// TwinCAT 3 PLC project LF_System_PLC
// ProgramVersion: 3.1.4026.20
// CompilerDefines: VISU_USEPROPERTYINFO
// libraries:
//   Tc2_Standard, * (Beckhoff Automation GmbH)
//   Tc2_System, * (Beckhoff Automation GmbH)
//   VisuSymbols, 4.5.0.0 (System)
// project tree:
//   DUTs/ Betriebszustand.TcDUT (not stored)
//   / GlobalTextList.TcGTLO, PlcTask.TcTTO (not stored), Visualization Manager.TcVMO (not stored)
//   POUs/Extruder/ FB_System_FlaschenFullstand.TcPOU (not stored), FB_System_Fullstand.TcPOU (not stored)
//   POUs/Förderband/ FB_System_CNV.TcPOU
//   POUs/ MAIN.TcPOU
//   POUs/Manipulator/ FB_System_LinAxis.TcPOU (not stored)
//   POUs/Vereinzelung/ FB_SpeicherRohr.TcPOU (not stored), FB_System_Vereinzelung.TcPOU (not stored)
//   VISUs/ Visualization.TcVIS
// (motion and I/O tree: see PLC project tempmodel)
// real-time tasks:
//   TASK PlcTask: cycle T#10ms, priority 21, ADS port 350
//   TASK PlcTask1: cycle T#10ms, priority 22, ADS port 351
//   TASK PlcTask2: cycle T#10ms, priority 20, ADS port 352
// variable links:
//   LF_System_PLC/LF_System_PLC Instance <-> NC-Task 1 SAF/Axes/BandAchse
//     PlcTask Inputs/MAIN.fIN_CnvPos <-> Outputs/ToPlc/ActPos
//   LF_System_PLC/LF_System_PLC Instance <-> NC-Task 1 SAF/Axes/Extruder1
//     PlcTask Inputs/MAIN.fIN_ExtPos1 <-> Outputs/ToPlc/ActPos
//   LF_System_PLC/LF_System_PLC Instance <-> NC-Task 1 SAF/Axes/Extruder2
//     PlcTask Inputs/MAIN.fIN_ExtPos2 <-> Outputs/ToPlc/ActPos
//   LF_System_PLC/LF_System_PLC Instance <-> NC-Task 1 SAF/Axes/Extruder3
//     PlcTask Inputs/MAIN.fIN_ExtPos3 <-> Outputs/ToPlc/ActPos
//   LF_System_PLC/LF_System_PLC Instance <-> PLC/PLC Instance
//     PlcTask Inputs/MAIN.bIN_Gripper <-> PlcTask Outputs/IFC_HW.bGripperClosed
//     PlcTask Inputs/MAIN.bIN_Stopper1 <-> PlcTask Outputs/IFC_HW.bBandHub1
//     PlcTask Inputs/MAIN.bIN_Stopper2 <-> PlcTask Outputs/IFC_HW.bBandHub2
//     PlcTask Inputs/MAIN.bIN_Stopper3 <-> PlcTask Outputs/IFC_HW.bBandHub3
//     PlcTask Inputs/MAIN.bIn_LedGreen <-> PlcTask Outputs/IFC_HW.bAmpelGrun
//     PlcTask Inputs/MAIN.bIn_LedRot <-> PlcTask Outputs/IFC_HW.bAmpelRot
//     PlcTask Inputs/MAIN.bIn_LedYellow <-> PlcTask Outputs/IFC_HW.bAmpelGelb
//     PlcTask Inputs/MAIN.bIn_Schleuse1_L1 <-> PlcTask Outputs/IFC_HW.bR1AKT1
//     PlcTask Inputs/MAIN.bIn_Schleuse1_L2 <-> PlcTask Outputs/IFC_HW.bR2AKT1
//     PlcTask Inputs/MAIN.bIn_Schleuse2_L1 <-> PlcTask Outputs/IFC_HW.bR1AKT2
//     PlcTask Inputs/MAIN.bIn_Schleuse2_L2 <-> PlcTask Outputs/IFC_HW.bR2AKT2
//     PlcTask Outputs/MAIN.bEnable <-> PlcTask Inputs/IFC_HW.bEnable
//     PlcTask Outputs/MAIN.bExecute <-> PlcTask Inputs/IFC_HW.bExecute
//     PlcTask Outputs/MAIN.bOUT_CnvNS{1..4} <-> PlcTask Inputs/IFC_HW.bBandSens{1..4}  (4 links)
//     PlcTask Outputs/MAIN.bOut_VereinzelungNS1 <-> PlcTask Inputs/IFC_HW.bEinzelSens1
//     PlcTask Outputs/MAIN.bOut_VereinzelungNS2 <-> PlcTask Inputs/IFC_HW.bEinzelSens2
//     PlcTask Outputs/MAIN.bOut_VereinzelungNS3 <-> PlcTask Inputs/IFC_HW.bEinzelSens3

// ---- POUs/Förderband/FB_System_CNV.TcPOU
FUNCTION_BLOCK FB_System_CNV
VAR_INPUT
	fPos : LREAL;
	bStopper1 : BOOL;
	bStopper2 : BOOL;
	bStopper3 : BOOL;
	bBottleDropped : BOOL; 
END_VAR
VAR_OUTPUT
	bNS1 : BOOL;
	bNS2 : BOOL;
	bNS3 : BOOL;
	bNS4 : BOOL;
	bBottleLeft : BOOL;
END_VAR
VAR
	fBottlePos : LREAL; // Reale Position der Flasche
	iBottlePos : LREAL; // Visualisierungs Position der Flaschen
	bBottleMoving : BOOL; // Flasche kann sich Bewegen, kein Stopper geschlossen und Stopper Pos erreicht
	fOffPos : LREAL; // OffsetPos nach Bewegungsfreigabe durch Stopper rückzug...
	rTrigBottleMoving : R_Trig;
	rTrigBottleDropped : R_Trig;
	fStopperPos1 : LREAL := 125.0;
	fStopperPos2 : LREAL := 250.0;
	fStopperPos3 : LREAL := 375.0;
	fStopperPos4 : LREAL := 630.0;; // Ende des Förderbandes
	onTimerCNVClear : TON;
	bBottleOnCNV : BOOL;
	bCNVisMoving : BOOL;
	fPosAlt : LReal;
END_VAR

onTimerCNVClear(PT := T#1S);
rTrigBottleMoving(CLK := bBottleMoving);
rTrigBottleDropped(CLK := bBottleDropped);
IF rTrigBottleDropped.Q THEN
	bBottleOnCNV := TRUE;
END_IF
// Flaschen Position bestimmen
IF rTrigBottleMoving.Q OR rTrigBottleDropped.Q THEN
	fOffPos := fPos-fBottlePos;
END_IF
IF bBottleMoving AND bBottleOnCNV THEN
	fBottlePos := fPos-fOffPos;
END_IF
// Skalierungsfunktion für fBottlePos zu iBottlePos (Real zu Visualisierung)

iBottlePos := TO_INT(fBottlePos * 0.7);

// Bewegungsfreigabe
IF NOT bStopper1 AND fBottlePos > fStopperPos1 - 2.0 AND fBottlePos < fStopperPos1 + 2.0 THEN
	bBottleMoving := FALSE;
ELSIF NOT bStopper2 AND fBottlePos > fStopperPos2 - 2.0 AND fbottlePos < fStopperPos2 + 2.0 THEN
	bBottleMoving := FALSE;
ELSIF NOT bStopper3 AND fBottlePos > fStopperPos3 - 2.0 AND fBottlePos < fStopperPos3 + 2.0 THEN
	bBottleMoving := FALSE;
ELSIF fBottlePos > fStopperPos4 - 1.0 THEN
	bBottleMoving := FALSE;
ELSE
	bBottleMoving := TRUE;
END_IF
// Sensor aktivierung
// bNS1
IF fBottlePos > fStopperPos1 - 15.0 AND fBottlePos < fStopperPos1 + 5.0 THEN
	bNS1 := TRUE;
ELSE
	bNS1 := FALSE;
END_IF
//bNS2
IF fBottlePos > fStopperPos2 - 15.0 AND fBottlePos < fStopperPos2 + 5.0 THEN
	bNS2 := TRUE;
ELSE
	bNS2 := FALSE;
END_IF
//bNS3
IF fBottlePos > fStopperPos3 - 15.0 AND fBottlePos < fStopperPos3 + 5.0 THEN
	bNS3 := TRUE;
ELSE
	bNS3 := FALSE;
END_IF
//bNS4
IF fBottlePos > fStopperPos4 - 15.0 AND fBottlePos < fStopperPos4 + 5.0 THEN
	bNS4 := TRUE;
ELSE
	bNS4 := FALSE;
END_IF

// END of CNV, Clear after 1 sec.
bBottleLeft := False;
IF bNS4 THEN
	onTimerCNVClear.IN := TRUE;
	IF onTimerCNVClear.Q THEN
		fBottlePos := 0.0;
		onTimerCNVClear.IN := FALSE;
		bBottleOnCNV := FALSE;
		bBottleLeft := TRUE;
	END_IF
END_IF

// is CNV Moving?
IF fPosAlt < fPos THEN
	bCNVisMoving := TRUE;
ELSE
	bCNVisMoving := FALSE;
END_IF
fPosAlt := fPos;

END_FUNCTION_BLOCK

// ---- POUs/MAIN.TcPOU
PROGRAM MAIN
VAR
// Systemeingangssignale (Stellsignale für Aktoren)
	bEnable AT%Q* : BOOL;
	bExecute AT%Q* : BOOL;
	// Status Lampe
	bIn_LedRot 		AT%I* : BOOL;
	bIn_LedYellow 	AT%I* : BOOL;
	bIn_LedGreen 	AT%I* : BOOL;
	// Vereinzelung 
	bIn_Schleuse1_L1 AT%I* : BOOL; // + Öffnen - Schließen
	bIn_Schleuse1_L2 AT%I* : BOOL; // + Schließen - Öffnen
	bIn_Schleuse2_L1 AT%I* : BOOL; // + Öffnen - Schließen
	bIn_Schleuse2_L2 AT%I* : BOOL; // + Schließen - Öffnen
	// Förderband
	fIN_CnvPos AT%I* : LREAL;
	bIN_Stopper1 AT%I* : BOOL;
	bIN_Stopper2 AT%I* : BOOL;
	bIN_Stopper3 AT%I* : BOOL;
	// Extruder
	fIN_ExtPos1 AT%I* : LREAL;
	fIN_ExtPos2 AT%I* : LREAL;
	fIN_ExtPos3 AT%I* : LREAL;
	// Manipulator
	fIN_ManXPos AT%I* : LREAL;
	bIN_Gripper AT%I* : BOOL;
	
// Systemausgangssignale (Sensorsignale)
	//Vereinzelung
	bOut_VereinzelungNS1 AT%Q* : BOOL; // Flasche am Kopf
	bOut_VereinzelungNS2 AT%Q* : BOOL; // Flasche im Speicher
	bOut_VereinzelungNS3 AT%Q* : BOOL; // Flasche in Kammer
	//Förderband
	bOUT_CnvNS1 AT%Q* : BOOL;
	bOUT_CnvNS2 AT%Q* : BOOL;
	bOUT_CnvNS3 AT%Q* : BOOL;
	bOUT_CnvNS4 AT%Q* : BOOL;
	// Füllstandssensoren
	iOut_USS1 AT%Q* : UINT;
	iOut_USS2 AT%Q* : UINT;
	iOut_USS3 AT%Q* : UINT;
	// Manipulator
	bOUT_SensMinX AT%Q* : BOOL;
	bOUT_SensMaxX AT%Q* : BOOL;
	
// System FB
	fbVereinzelung : FB_System_Vereinzelung;	
	fbCNV : FB_System_CNV;
	fbExt1 : FB_System_Fullstand;
	fbExt2 : FB_System_Fullstand;
	fbExt3 : FB_System_Fullstand;
	fbBottleLevel : FB_System_FlaschenFullstand;
	fbManAxX : FB_System_LinAxis;
		
// Hilfsvariablen
	bRefill1 : BOOL;
	bRefill2 : BOOL;
	bRefill3 : BOOL;
	
	PosSensMinX : INT := 620;
	PosSensMaxX : INT := 1137;
END_VAR

fbVereinzelung(
	bS1L1:= bIn_Schleuse1_L1, 
	bS1L2:= bIn_Schleuse1_L2, 
	bS2L1:= bIn_Schleuse2_L1, 
	bS2L2:= bIn_Schleuse2_L2,
	bNS1=> bOut_VereinzelungNS1, 
	bNS2=> bOut_VereinzelungNS2, 
	bNS3=> bOut_VereinzelungNS3,
	bBottleDropped => );
	
fbCNV(
	fPos:= fIN_CnvPos, 
	bStopper1:= bIN_Stopper1, 
	bStopper2:= bIN_Stopper2, 
	bStopper3:= bIN_Stopper3, 
	bBottleDropped := fbVereinzelung.bBottleDropped , 
	bNS1=> bOut_CnvNS1 , 
	bNS2=> bOut_CnvNS2 , 
	bNS3=> bOut_CnvNS3 , 
	bNS4=> bOut_CnvNS4,
	bBottleLeft => );
	
fbExt1(bRefill:=bRefill1 , fPosExt:= fIN_ExtPos1, iOut=> iOut_USS1 );
fbExt2(bRefill:=bRefill2 , fPosExt:= fIN_ExtPos2, iOut=> iOut_USS2 );
fbExt3(bRefill:=bRefill3 , fPosExt:= fIN_ExtPos3, iOut=> iOut_USS3 );

fbBottleLevel(rFilling1 := fIN_ExtPos1, rFilling2 := fIN_ExtPos2 ,rFilling3 := fIN_ExtPos3,Reset:= fbCNV.bBottleDropped );

fbManAxX(fPos := fIN_ManXPos,
		bGripperOpen := bIN_Gripper,
		bSensMin => bOut_SensMinX,
		bSensMax => bOut_SensMaxX, 
		);

END_PROGRAM

// ---- GlobalTextList.TcGTLO
TEXTLIST GlobalTextList
  477 = 'Befüllen'
  647 = 'Enable'
  925 = 'Execute'
  401 = 'X'
END_TEXTLIST

// ---- VISUs/Visualization.TcVIS
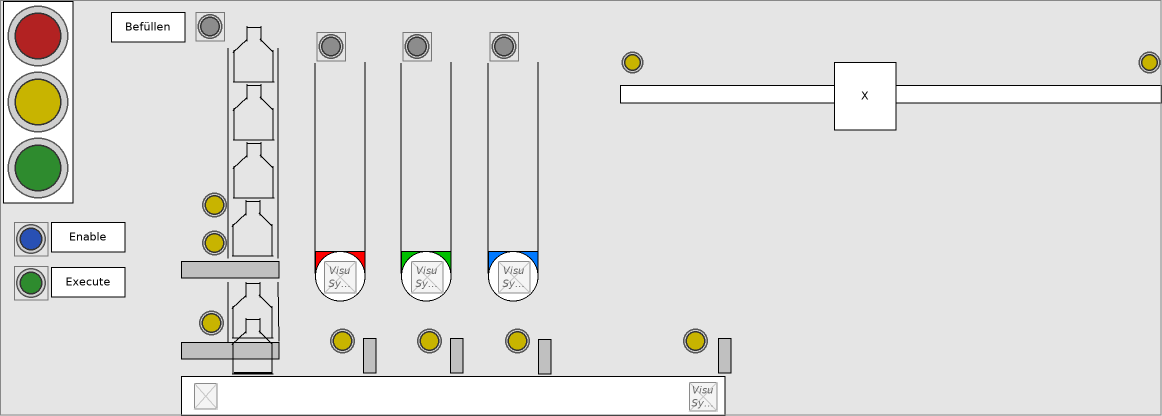
VISUALIZATION Visualization  // 1162x416
    Rectangle (315,251 50x24)
        p2773130477: - MAIN.fbExt1.iFillLevel
    Lamp1 (200,190 29x30), variable: MAIN.bOut_VereinzelungNS1, style: Lamp-Lamp1-Yellow
    Lamp1 (200,228 29x30), variable: MAIN.bOut_VereinzelungNS2, style: Lamp-Lamp1-Yellow
    Lamp1 (197,308 29x30), variable: MAIN.bOut_VereinzelungNS3, style: Lamp-Lamp1-Yellow
    Group (3,1 70x202)
        Rectangle (0,0 70x202)
        Lamp1 (0,0 70x70), variable: MAIN.bIn_LedRot, style: Lamp-Lamp1-Red
        Lamp1 (0,66 70x70), variable: MAIN.bIn_LedYellow, style: Lamp-Lamp1-Yellow
        Lamp1 (0,132 70x70), variable: MAIN.bIn_LedGreen, style: Lamp-Lamp1-Green
    Line (228,258) (228,48)
    Line (278,258) (278,48)
    Line (279,341) (278,282)
    Line (228,342) (228,282)
    Rectangle (181,261 98x17)
        p3528305787: MAIN.fbVereinzelung.S1pos
        p874137650: MAIN.fbVereinzelung.S1pos
    Rectangle (181,342 98x17)
        p3528305787: MAIN.fbVereinzelung.S2pos
        p874137650: MAIN.fbVereinzelung.S2pos
    PushSwitch (12,222 38x34), variable: MAIN.bEnable, behaviour: TOGGLE, style: Switch-PushSwitch-Blue
    PushSwitch (12,266 38x34), variable: MAIN.bExecute, behaviour: TAP, style: Switch-PushSwitch-Green
    Rectangle (51,222 74x30), "Enable"
    Rectangle (51,267 74x30), "Execute"
    Group (232,200 41x57), invisible if: not MAIN.fbVereinzelung.fbSpeicherRohr.aSpeicher[0]
        Line (1,56) (1,24)
        Line (40,55) (40,24)
        Line (41,56) (0,56)
        Line (0,26) (14,13)
        Line (40,26) (27,13)
        Line (14,15) (14,0)
        Line (28,15) (28,0)
        Line (14,1) (28,1)
    Group (233,142 41x57), invisible if: Not MAIN.fbVereinzelung.fbSpeicherRohr.aSpeicher[1]
        Line (1,56) (1,24)
        Line (40,55) (40,24)
        Line (41,56) (0,56)
        Line (0,26) (14,13)
        Line (40,26) (27,13)
        Line (14,15) (14,0)
        Line (28,15) (28,0)
        Line (14,1) (28,1)
    Group (232,282 41x57), invisible if: not MAIN.bOut_VereinzelungNS3
        Line (1,56) (1,24)
        Line (40,55) (40,24)
        Line (41,56) (0,56)
        Line (0,26) (14,13)
        Line (40,26) (27,13)
        Line (14,15) (14,0)
        Line (28,15) (28,0)
        Line (14,1) (28,1)
    Group (233,84 41x57), invisible if: Not MAIN.fbVereinzelung.fbSpeicherRohr.aSpeicher[2]
        Line (1,56) (1,24)
        Line (40,55) (40,24)
        Line (41,56) (0,56)
        Line (0,26) (14,13)
        Line (40,26) (27,13)
        Line (14,15) (14,0)
        Line (28,15) (28,0)
        Line (14,1) (28,1)
    Group (233,26 41x57), invisible if: Not MAIN.fbVereinzelung.fbSpeicherRohr.aSpeicher[3]
        Line (1,56) (1,24)
        Line (40,55) (40,24)
        Line (41,56) (0,56)
        Line (0,26) (14,13)
        Line (40,26) (27,13)
        Line (14,15) (14,0)
        Line (28,15) (28,0)
        Line (14,1) (28,1)
    PushSwitch (194,12 32x29), variable: MAIN.fbVereinzelung.bBefullen, behaviour: TAP, style: Switch-PushSwitch-Gray
    RoundedRectangle (181,376 544x40)
    Lamp1 (328,326 29x30), variable: MAIN.bOUT_CnvNS1, style: Lamp-Lamp1-Yellow
    Lamp1 (503,326 29x30), variable: MAIN.bOUT_CnvNS3, style: Lamp-Lamp1-Yellow
    Lamp1 (415,326 29x30), variable: MAIN.bOUT_CnvNS2, style: Lamp-Lamp1-Yellow
    Lamp1 (681,326 29x30), variable: MAIN.bOUT_CnvNS4, style: Lamp-Lamp1-Yellow
    Group (232,318 41x57), invisible if: not MAIN.fbCNV.bBottleOnCNV
        p3560616238: MAIN.fbCNV.iBottlePos
        Line (1,56) (1,24)
        Line (40,55) (40,24)
        Line (41,56) (0,56)
        Line (0,26) (14,13)
        Line (40,26) (27,13)
        Line (14,15) (14,0)
        Line (28,15) (28,0)
        Line (14,1) (28,1)
    Rectangle (363,338 13x35), invisible if: MAIN.bIN_Stopper1
    Rectangle (450,338 13x35), invisible if: MAIN.bIN_Stopper2
    Rectangle (538,339 13x35), invisible if: MAIN.bIN_Stopper3
    Rectangle (718,338 13x35)
    Image (194,383 23x26), invisible if: not MAIN.fbCNV.bCNVisMoving, image: VisuSymbols.Symbols.ArrowHalfRightUp
    Image (689,382 28x29), invisible if: not MAIN.fbCNV.bCNVisMoving, image: VisuSymbols.Symbols.ArrowHalfRightDown
    Rectangle (111,12 74x30), "Befüllen"
    Ellipse (315,251 50x50)
    Line (315,273) (315,63)
    Line (365,272) (365,62)
    Rectangle (401,251 50x24)
        p2773130477: - MAIN.fbExt2.iFillLevel
    Ellipse (401,251 50x50)
    Line (401,273) (401,63)
    Line (451,272) (451,62)
    Rectangle (488,251 50x24)
        p2773130477: - MAIN.fbExt3.iFillLevel
    Ellipse (488,251 50x50)
    Line (488,273) (488,63)
    Line (538,272) (538,62)
    PushSwitch (315,32 32x29), variable: MAIN.bRefill1, behaviour: TAP, style: Switch-PushSwitch-Gray
    PushSwitch (401,32 32x29), variable: MAIN.bRefill2, behaviour: TAP, style: Switch-PushSwitch-Gray
    PushSwitch (488,32 32x29), variable: MAIN.bRefill3, behaviour: TAP, style: Switch-PushSwitch-Gray
    Image (324,261 32x32), invisible if: MAIN.fbExt1.NotMoving, image: VisuSymbols.Symbols.ArrowCircle2RightRightLeft
    Image (411,261 32x32), invisible if: MAIN.fbExt2.NotMoving, image: VisuSymbols.Symbols.ArrowCircle2RightRightLeft
    Image (498,261 32x32), invisible if: MAIN.fbExt3.NotMoving, image: VisuSymbols.Symbols.ArrowCircle2RightRightLeft
    Rectangle (234,372 38x1), invisible if: not MAIN.fbCNV.bBottleOnCNV
        p2773130477: - MAIN.fbBottleLevel.iFillLevel3 - MAIN.fbBottleLevel.iFillLevel1 - MAIN.fbBottleLevel.iFillLevel2
        p3560616238: MAIN.fbCNV.iBottlePos
        p1126004900: - MAIN.fbBottleLevel.iFillLevel1 - MAIN.fbBottleLevel.iFillLevel2
    Rectangle (234,372 38x1), invisible if: not MAIN.fbCNV.bBottleOnCNV
        p2773130477: - MAIN.fbBottleLevel.iFillLevel2 - MAIN.fbBottleLevel.iFillLevel1
        p3560616238: MAIN.fbCNV.iBottlePos
        p1126004900: - MAIN.fbBottleLevel.iFillLevel1
    Rectangle (234,372 38x1), invisible if: not MAIN.fbCNV.bBottleOnCNV
        p2773130477: - MAIN.fbBottleLevel.iFillLevel1
        p3560616238: MAIN.fbCNV.iBottlePos
    Rectangle (620,85 542x18)
    Rectangle (834,62 62x68), "X"
        p3560616238: MAIN.fbManAxX.iAxPos
    Lamp1 (620,50 25x25), variable: MAIN.bOUT_SensMinX, style: Lamp-Lamp1-Yellow
    Lamp1 (1137,50 25x25), variable: MAIN.bOUT_SensMaxX, style: Lamp-Lamp1-Yellow
END_VISUALIZATION
